Universal Robots PolyScope program: sprayFront.urp

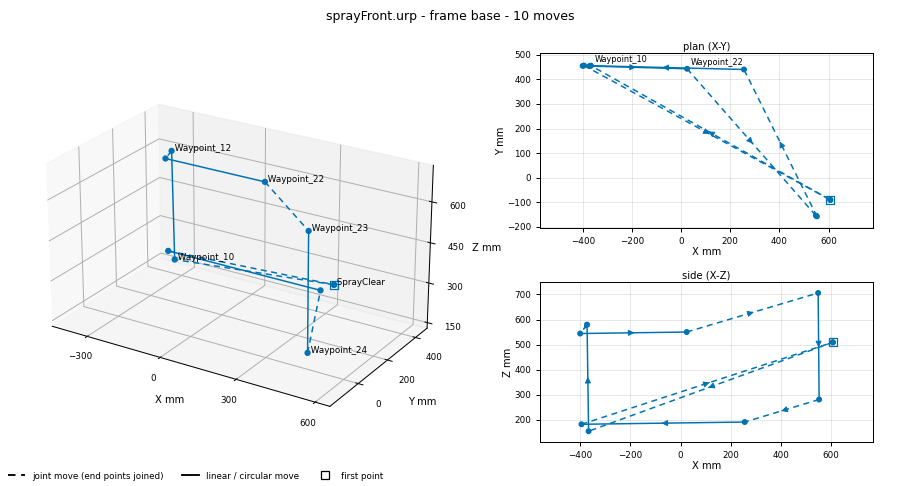
[picture p0: tool path of sprayFront.urp in frame base, 10 of 10 moves have a stored position in this frame; points joined in program order, loops and branches not executed]
Program sprayFront (installation=sand5 directory=/programs/subs createdIn=5.11.5.1010327 lastSavedIn=5.11.5.1010327 robotSerialNumber=20215500677)
Calibrated DH parameters: a=[0.000204, -0.239222, -0.391845, -0.000001, 0.000022, 0]; d=[0.162722, -355.808559, 353.37206, 2.570385, 0.099741, 0.099629]; alpha=[1.571124, 0.000988, 0.008295, 1.568963, -1.570303, 0]; deltaTheta=[0, -0.973091, 7.204745, 0.05153, 0, 0]
Robot Program (runOnlyOnce=false)
  Folder SprayFront
    MoveJ speed 60 deg/s, acceleration 80 deg/s^2 (useActiveTCP=false) tcp=Spray; feature=SprayPlane
      Waypoint SprayClear: TCP in base x=607.137 y=-90.197 z=509.102 mm, rx=1.2034 ry=1.2067 rz=1.2159 rad; joints [154.541, -56.922, 94.352, -266.679, -69.476, 23.135] deg; TCP offset x=20.839 y=-27.14 z=105.994 mm, rx=0.1226 ry=1.1769 rz=2.8697 rad; feature pose in base x=807.673 y=110.818 z=310.566 mm, rx=1.2166 ry=-1.2106 rz=-1.2041 rad
    MoveJ speed 60 deg/s, acceleration 80 deg/s^2 (useActiveTCP=false) tcp=Spray; feature=SprayPlane
      Waypoint Waypoint_10: TCP in base x=-366.88 y=455.74 z=154.683 mm, rx=-1.1923 ry=1.2085 rz=1.1804 rad; joints [282.195, -40.36, 126.156, -261.512, -59.605, -89.075] deg; TCP offset x=20.839 y=-27.14 z=105.994 mm, rx=0.1226 ry=1.1769 rz=2.8697 rad; feature pose in base x=-366.784 y=580.679 z=180.17 mm, rx=1.5749 ry=-0.0329 rz=-0.0106 rad
      Set DigitalOutput pin=digital_out[4]; digitalValue=1
    MoveL speed 100 mm/s, acceleration 1200 mm/s^2 (useActiveTCP=true) feature=SprayPlane
      Waypoint Waypoint_12: TCP in base x=-372.961 y=453.99 z=579.608 mm, rx=-1.1924 ry=1.2084 rz=1.1805 rad; joints [283.1, -92.847, 109.867, -192.963, -60.146, -88.612] deg
      Set DigitalOutput pin=digital_out[4]; digitalValue=0
      MoveDirectionNode (selectedDirection=ZMinus toolParams=0.2, 1.2) feature=Joint_6_name
        Until DISTANCE (allowActions=false deceleration=3 distanceNodeType=STOP) Distance=0.1; motionParameters(blendRadius=0)
    MoveJ speed 60 deg/s, acceleration 80 deg/s^2 (useActiveTCP=false) tcp=Spray; feature=SprayPlane
      Waypoint Waypoint_21: TCP in base x=-400.443 y=454.966 z=544.225 mm, rx=-1.5663 ry=0.0105 rz=-0.0329 rad; joints [305.438, -86.323, 77.292, -117.871, -118.512, -147.771] deg
      Set DigitalOutput pin=digital_out[4]; digitalValue=1
    MoveL speed 100 mm/s, acceleration 1200 mm/s^2 (useActiveTCP=false) tcp=Spray; feature=SprayPlane
      Waypoint Waypoint_22: TCP in base x=24.363 y=443.181 z=550.193 mm, rx=-1.5664 ry=0.0106 rz=-0.0328 rad; joints [239.529, -113.419, 99.688, -119.587, -73.088, -197.229] deg
      Set DigitalOutput pin=digital_out[4]; digitalValue=0
      MoveDirectionNode (selectedDirection=ZMinus toolParams=0.2, 1.2) feature=Joint_6_name
        Until DISTANCE (allowActions=false deceleration=3 distanceNodeType=STOP) Distance=0.1; motionParameters(blendRadius=0)
    MoveJ speed 60 deg/s, acceleration 80 deg/s^2 (useActiveTCP=false) tcp=Spray; feature=SprayPlane
      Waypoint Waypoint_23: TCP in base x=548.641 y=-154.61 z=706.095 mm, rx=-0.0121 ry=1.5616 rz=0.002 rad; joints [128.296, -68.562, 32.652, 13.403, -7.79, -244.639] deg; TCP offset x=20.839 y=-27.14 z=105.994 mm, rx=0.1226 ry=1.1769 rz=2.8697 rad; feature pose in base x=674.096 y=208.92 z=304.834 mm, rx=1.2154 ry=-1.2124 rz=-1.1935 rad
      Set DigitalOutput pin=digital_out[4]; digitalValue=1
    MoveL speed 100 mm/s, acceleration 1200 mm/s^2 (useActiveTCP=false) tcp=Spray; feature=SprayPlane
      Waypoint Waypoint_24: TCP in base x=552.545 y=-157.368 z=281.062 mm, rx=-0.0121 ry=1.5615 rz=0.0019 rad; joints [128.403, -70.766, 101.674, -54.987, -7.187, -243.057] deg
      Set DigitalOutput pin=digital_out[4]; digitalValue=0
      MoveDirectionNode (selectedDirection=ZMinus toolParams=0.2, 1.2) feature=Joint_6_name
        Until DISTANCE (allowActions=false deceleration=3 distanceNodeType=STOP) Distance=0.1; motionParameters(blendRadius=0)
      MoveDirectionNode (selectedDirection=ZPlus) feature=Base
        Until DISTANCE (allowActions=false deceleration=3 distanceNodeType=STOP) Distance=0.1; motionParameters(blendRadius=0)
    MoveJ speed 60 deg/s, acceleration 80 deg/s^2 (useActiveTCP=false) tcp=Spray; feature=SprayPlane
      Waypoint Waypoint_38: TCP in base x=255.883 y=440.293 z=191.235 mm, rx=-1.5741 ry=0.008 rz=-0.0287 rad; joints [210.744, -86.11, 132.363, -168.194, -55.616, -222.536] deg; TCP offset x=20.839 y=-27.14 z=105.994 mm, rx=0.1226 ry=1.1769 rz=2.8697 rad; feature pose in base x=-141.025 y=574.651 z=182.515 mm, rx=1.5672 ry=-0.0288 rz=-0.0081 rad
      Set DigitalOutput pin=digital_out[4]; digitalValue=1
    MoveL speed 100 mm/s, acceleration 1200 mm/s^2 (useActiveTCP=false) tcp=Spray; feature=SprayPlane
      Waypoint Waypoint_25: TCP in base x=-395.272 y=456.409 z=182.261 mm, rx=-1.5664 ry=0.0105 rz=-0.0328 rad; joints [304.782, -71.234, 116.575, -172.386, -118.444, -148.069] deg; TCP offset x=20.839 y=-27.14 z=105.994 mm, rx=0.1226 ry=1.1769 rz=2.8697 rad; feature pose in base x=-366.784 y=580.679 z=180.17 mm, rx=1.5749 ry=-0.0329 rz=-0.0106 rad
      Set DigitalOutput pin=digital_out[4]; digitalValue=0
      MoveDirectionNode (selectedDirection=ZMinus toolParams=0.2, 1.2) feature=Joint_6_name
        Until DISTANCE (allowActions=false deceleration=3 distanceNodeType=STOP) Distance=0.1; motionParameters(blendRadius=0)
    MoveJ speed 60 deg/s, acceleration 80 deg/s^2 (useActiveTCP=false) tcp=Spray; feature=SprayPlane
      Waypoint SprayClear: TCP in base x=607.137 y=-90.197 z=509.102 mm, rx=1.2034 ry=1.2067 rz=1.2159 rad; joints [154.541, -56.922, 94.352, -266.679, -69.476, 23.135] deg; TCP offset x=20.839 y=-27.14 z=105.994 mm, rx=0.1226 ry=1.1769 rz=2.8697 rad; feature pose in base x=807.673 y=110.818 z=310.566 mm, rx=1.2166 ry=-1.2106 rz=-1.2041 rad
